TYPE ST_MainSequencerStatus :
STRUCT
	PowerOn 		: BOOL;
	ResetRequired	: BOOL;
	Auto			: BOOL;
	MaintenanceMode	: BOOL;
END_STRUCT
END_TYPE

(* stored: Version 1.1.0.1, ProductVersion 3.1.4024.12
   DUT ST_MainSequencerStatus: Id {718a9102-6ecf-4ddd-bcd2-48348f2ffe1d} *)
